FUNCTION_BLOCK PUBLIC AutomaticControl
VAR_INPUT
    Switch: BOOL;
END_VAR
VAR
    State: INT := 0;
    ExecutingRecipe1: BOOL := FALSE;
    ExecutingRecipe2: BOOL := FALSE;
	myRecipe1: Recipe1;
    myRecipe2: Recipe2;
    Tmp: BOOL;
    RestorePreviousAutomaticState: RestorePreviousAutomaticState;
	CountCurrentPosition1: CountCurrentPosition1;
	Safety: Safety1;
END_VAR
VAR_OUTPUT
    Output: BOOL := TRUE;
END_VAR

// TwinCAT ensures that all POUs, including your AutomaticControl program 
// and Recipe1() Function Block, are executed once per cycle.

// for debugging purposes:
IF IO.ButtonRed THEN
	IO.Initialized := FALSE;
END_IF


IF (NOT IO.Initialized) THEN
	Initialize();
ELSIF (NOT IO.Switch) AND IO.PreviousManualMode THEN
	CountCurrentPosition1();
	Safety();
	RestorePreviousAutomaticState();
ELSE
	CountCurrentPosition1();
	Safety();
	
    IF (IO.ButtonUpperLeft OR ExecutingRecipe1) AND Automatic.AllRestored THEN
        myRecipe1.ExecutingRecipe1 := TRUE;
		myRecipe1();
		myRecipe1.SuccesfullyEnded1 := FALSE;
		ExecutingRecipe1 := NOT myRecipe1.SuccesfullyEnded;
    ELSIF (NOT ExecutingRecipe1) AND (IO.ButtonUpperRight OR ExecutingRecipe2) AND Automatic.AllRestored THEN
        myRecipe2.ExecutingRecipe2 := TRUE; // Pass input to the function block
        myRecipe2(); // Call the function block
		myRecipe2.SuccesfullyEnded2 := FALSE;
        ExecutingRecipe2 := NOT myRecipe2.SuccesfullyEnded;
    END_IF
END_IF




RETURN;

END_FUNCTION_BLOCK

(* stored: Version 1.1.0.1, ProductVersion 3.1.4024.13
   POU AutomaticControl: Id {f9244839-88dd-4f0f-95ab-d4274120fb90}, SpecialFunc None *)
